PROGRAM MAIN
VAR
END_VAR

timer := timer + 0.01;

END_PROGRAM

(* stored: Version 1.1.0.1, ProductVersion 3.1.0.38
   POU MAIN: Id {29a53d6f-2791-434c-ac0e-95c286c60a9e}, SpecialFunc None *)
